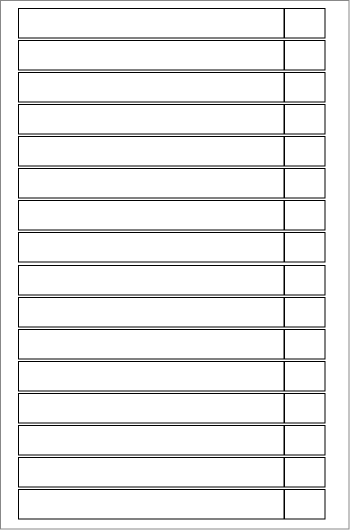
VISUALIZATION Vis_Interlock_base  // 350x530
VAR_IN_OUT
	stHMIInterlock:stHMI_Interlock;
END_VAR
    Rectangle (18,8 266x30), text variable: stHMIInterlock.asInterlockNames[1]
    Rectangle (284,8 41x30), colour toggle: stHMIInterlock.abInterlocks[1]
    Rectangle (18,40 266x30)
    Rectangle (284,40 41x30)
    Rectangle (18,72 266x30)
    Rectangle (284,72 41x30)
    Rectangle (18,104 266x30)
    Rectangle (284,104 41x30)
    Rectangle (18,136 266x30)
    Rectangle (284,136 41x30)
    Rectangle (18,168 266x30)
    Rectangle (284,168 41x30)
    Rectangle (18,200 266x30)
    Rectangle (284,200 41x30)
    Rectangle (18,232 266x30)
    Rectangle (284,232 41x30)
    Rectangle (18,265 266x30)
    Rectangle (284,265 41x30)
    Rectangle (18,297 266x30)
    Rectangle (284,297 41x30)
    Rectangle (18,329 266x30)
    Rectangle (284,329 41x30)
    Rectangle (18,361 266x30)
    Rectangle (284,361 41x30)
    Rectangle (18,393 266x30)
    Rectangle (284,393 41x30)
    Rectangle (18,425 266x30)
    Rectangle (284,425 41x30)
    Rectangle (18,457 266x30)
    Rectangle (284,457 41x30)
    Rectangle (18,489 266x30)
    Rectangle (284,489 41x30)
END_VISUALIZATION

(* stored: Version 1.1.0.1, ProductVersion 3.1.4024.11
   Visu Vis_Interlock_base: Id {99eefa14-c101-42b0-8990-39ec8d7de5f3} *)
